TYPE (* A Structure with 1 BOOL *)
  (* Version 1.0, 2024-02-21, Franz Höpfinger, HR Agrartechnik GmbH *)
  ST01B : STRUCT
    B_00 : BOOL; (* BIT 00 *)
  END_STRUCT;
END_TYPE
